{attribute 'GeneratedUsingTerminal: EK1122-0000-0018'}
{attribute addProperty BoxType "EK1122-0000-0018"}
{attribute addProperty Id "Beckhoff_ER8xxxsub_EK1100EK1100_1FC0878B2A_0001_ER8309_1022_0018ER8309_A0C54F7770"}
{attribute addProperty CRC "3438986324"}
{attribute addProperty Size "72"}
TYPE Beckhoff_ER8xxxEK1122_CCFAC454 EXTENDS EK1122_1FC0878B :
STRUCT
	{attribute addProperty Name "Beckhoff_ER8xxxsub_EK1100"}
	{attribute addProperty PreviousPort "Beckhoff ER8xxxEK1122 : D"}
	Beckhoff_ER8xxxsub_EK1100 : EK1100_1FC0878B;
	{attribute addProperty Name "A_0001_ER8309_1022_0018"}
	{attribute addProperty PreviousPort "Beckhoff ER8xxxsub EK1100 : C"}
	A_0001_ER8309_1022_0018 : ER8309_A0C54F77;
END_STRUCT
END_TYPE

(* stored: Version 1.2.0.0, ProductVersion 3.1.4024.9
   DUT Beckhoff_ER8xxxEK1122_CCFAC454: Id {df5596ec-7fe6-4770-b04d-6917397bb5f4} *)
